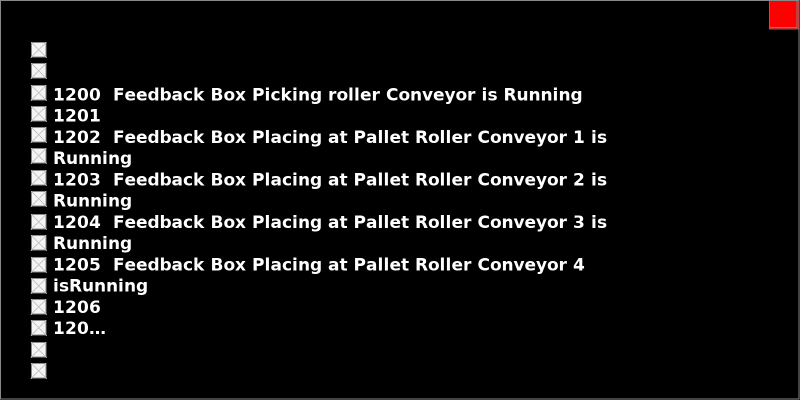
VISUALIZATION P1_DI2  // 800x400, background image 
    ImageSwitcher (31,42 15x15), variable: InputOutput_GVL.xIn1200, behaviour: TOGGLE
    Label (50,16 625x391), "1200 Feedback Box Picking roller Conveyor is Running 1201 1202 Feedback Box Placing at Pallet Roller Conveyor 1 is Running 1203 Feedback Box Placing at Pallet Roller Conveyor 2 is Running 1204 Feedback Box Placing at Pallet Roller Conveyor 3 is Running 1205 Feedback Box Placing at Pallet Roller Conveyor 4 isRunning 1206 1207 1208 1209 1210 1211 RSW Pneumatic Box Centring When Rtc 1212 RSW Pneumatic Gap Maker When Adv 1213 RSW Pneumatic Gap Maker When Rtc 1214 RSW Pneumatic Stopper Transfer When Rtc 1215"
    ImageSwitcher (31,63 15x15), variable: InputOutput_GVL.xIn1201, behaviour: TOGGLE
    ImageSwitcher (31,85 15x15), variable: InputOutput_GVL.xIn1202, behaviour: TOGGLE
    ImageSwitcher (31,106 15x15), variable: InputOutput_GVL.xIn1203, behaviour: TOGGLE
    ImageSwitcher (31,127 15x15), variable: InputOutput_GVL.xIn1204, behaviour: TOGGLE
    ImageSwitcher (31,148 15x15), variable: InputOutput_GVL.xIn1205, behaviour: TOGGLE
    ImageSwitcher (31,170 15x15), variable: InputOutput_GVL.xIn1206, behaviour: TOGGLE
    ImageSwitcher (31,191 15x15), variable: InputOutput_GVL.xIn1207, behaviour: TOGGLE
    ImageSwitcher (31,214 15x15), variable: InputOutput_GVL.xIn1208, behaviour: TOGGLE
    ImageSwitcher (31,235 15x15), variable: InputOutput_GVL.xIn1209, behaviour: TOGGLE
    ImageSwitcher (31,257 15x15), variable: InputOutput_GVL.xIn1210, behaviour: TOGGLE
    ImageSwitcher (31,278 15x15), variable: InputOutput_GVL.xIn1211, behaviour: TOGGLE
    ImageSwitcher (31,299 15x15), variable: InputOutput_GVL.xIn1212, behaviour: TOGGLE
    ImageSwitcher (31,320 15x15), variable: InputOutput_GVL.xIn1213, behaviour: TOGGLE
    ImageSwitcher (31,342 15x15), variable: InputOutput_GVL.xIn1214, behaviour: TOGGLE
    ImageSwitcher (31,363 15x15), variable: InputOutput_GVL.xIn1215, behaviour: TOGGLE
    Button (769,-1 30x30), image: VisuSymbols.Symbols.Wrong
        OnMouseClick: CloseDialog Dialog=P1_DI2, Result=OK, NumpadKeypadSet=True
END_VISUALIZATION

(* stored: Version 1.1.0.1, ProductVersion 3.1.4024.12
   Visu P1_DI2: Id {cff69a77-2e28-4bb6-b50a-0707f4d1d2c3} *)
